PROGRAM Logic
VAR
	FB_MBUS_EMH_DIZ_0: FB_MBUS_EMH_DIZ;
	FB_MBUSKL6781_0: FB_MBUSKL6781;
	mStart: BOOL;
	stComIn  AT%I*: ST_KL6781inData22B;
	stComOut AT%Q*: ST_KL6781outData22B;
	stCom    : ST_MBUS_Communication;
	mDisabled: BOOL;
	R_TRIG_0: r_trig;
	string_Error: E_MBUS_Error;
	string_Error_OK: E_MBUS_Error;
	mTriggered: BOOL;
END_VAR

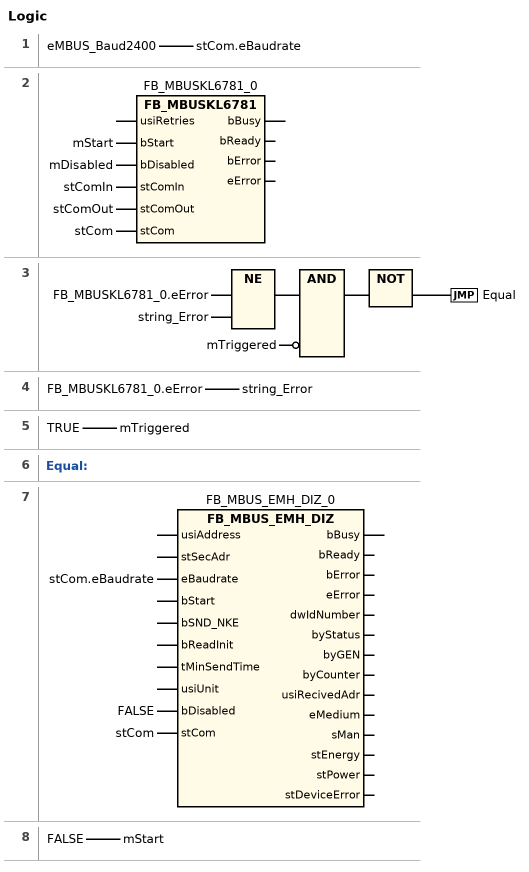
// NETWORK 1
stCom.eBaudrate := eMBUS_Baud2400;

// NETWORK 2
FB_MBUSKL6781_0(
    bStart := mStart,
    bDisabled := mDisabled,
    stComIn := stComIn,
    stComOut := stComOut,
    stCom := stCom); // FB_MBUSKL6781

// NETWORK 3
IF NOT (FB_MBUSKL6781_0.eError <> string_Error AND NOT mTriggered) THEN JMP Equal; END_IF

// NETWORK 4
string_Error := FB_MBUSKL6781_0.eError;

// NETWORK 5
mTriggered := TRUE;

// NETWORK 6
Equal: ;

// NETWORK 7
FB_MBUS_EMH_DIZ_0(eBaudrate := stCom.eBaudrate, bDisabled := FALSE, stCom := stCom); // FB_MBUS_EMH_DIZ

// NETWORK 8
mStart := FALSE;

END_PROGRAM

(* stored: Version 1.1.0.1, ProductVersion 3.1.4024.11
   POU Logic: Id {94017343-24fd-4b60-ba28-9ec8b681218b}, SpecialFunc None *)
